(* CODESYS project Elevator.ecp

Project tree, tasks and I/O mapping:
  Controller : 750-8214 PFC200 G2 2ETH RS CAN, WAGO, order no. 0750-8214, version 5.13.2.32
    application Application
      libraries: ; WagoAppPlcModbus, 1.1.2.3 (WAGO)
      task PLC_Task (cyclic, interval t#50ms, priority 15) calls ModbusTester, Heis2Test, VariableAssociation
      task VISU_TASK (cyclic, interval 100 ms, priority 15) calls VisuElems.Visu_Prg
      global variables GVL
      program ModbusTester [ST]
      MODBUS/
        data type typHeis1_tcp
        data type typHeis2_tcp
      global variables MODBUS
      program VariableAssociation [ST]
      program Heis2Test [ST]
      visualisation Visualization
    Kbus : Kbus, WAGO, version 1.4.0.2
        unmapped channels: K-BUS diagnostics
      _8_DI_Generic : 075x-8DI, WAGO, order no. 075x-8DI, version 0.0.0.13
          settings: K-BUS Module slot index = 1
          unmapped channels: _IN
      _8_DO_Generic : 075x-8DO, WAGO, order no. 075x-8DO, version 0.0.0.13
          settings: K-BUS Module slot index = 2
          unmapped channels: _OUT
    MODBUS
      MODBUS : MODBUS, WAGO, order no. n/a, version 1.1.1.15
        _internal_1006_0001_Master : MODBUS Master, WAGO, order no. n/a, version 1.1.1.15
          _internal_1006_0001_IP : MODBUS IP Interface, WAGO, order no. n/a, version 1.1.1.15
              settings: IP settings.Address = '192.168.0.3'
            Heis1_tcp : MODBUS Remote Slave, WAGO, order no. n/a, version 1.1.1.15
                settings: Channel100005.Priority = 1; Channel100005.Cycle Time = 200 ms; Channel100005.Read Length = 24 Registers or Coils; ChannelOffset100010 = 0; ChannelOffset100030 = 1; ChannelOffset100050 = 2; ChannelOffset100070 = 3; ChannelOffset100090 = 4; ChannelOffset100110 = 5; ChannelOffset100130 = 6; ChannelOffset100150 = 7; ChannelOffset100170 = 8; ChannelOffset100190 = 9; ChannelOffset100210 = 10; ChannelOffset100230 = 11; ChannelOffset100250 = 12; ChannelOffset100270 = 13; ChannelOffset100290 = 14; ChannelOffset100310 = 15; ChannelOffset100330 = 16; ChannelOffset100350 = 17; ChannelOffset100370 = 18; ChannelOffset100390 = 19; ChannelOffset100410 = 20; ChannelOffset100430 = 21; ChannelOffset100450 = 22; ChannelOffset100470 = 23; Channel100485.Priority = 1; Channel100485.Cycle Time = 200 ms; Channel100485.Write Address = 512 Registers or Coils; Channel100485.Write Length = 16 Registers or Coils; ChannelOffset100490 = 0; ChannelOffset100510 = 1; ChannelOffset100530 = 2; ChannelOffset100550 = 3; ChannelOffset100570 = 4; ChannelOffset100590 = 5; ChannelOffset100610 = 6; ChannelOffset100630 = 7; ChannelOffset100650 = 8;
                  ChannelOffset100670 = 9; ChannelOffset100690 = 10; ChannelOffset100710 = 11; ChannelOffset100730 = 12; ChannelOffset100750 = 13; ChannelOffset100770 = 14; ChannelOffset100790 = 15; Slave address / Unit identifier = 2
                input  Application.MODBUS.Heis1_tcp.dIn_1 : BOOL  // ChannelMapping100020
                input  Application.MODBUS.Heis1_tcp.dIn_2 : BOOL  // ChannelMapping100040
                input  Application.MODBUS.Heis1_tcp.dIn_3 : BOOL  // ChannelMapping100060
                input  Application.MODBUS.Heis1_tcp.dIn_4 : BOOL  // ChannelMapping100080
                input  Application.MODBUS.Heis1_tcp.dIn_5 : BOOL  // ChannelMapping100100
                input  Application.MODBUS.Heis1_tcp.dIn_6 : BOOL  // ChannelMapping100120
                input  Application.MODBUS.Heis1_tcp.dIn_7 : BOOL  // ChannelMapping100140
                input  Application.MODBUS.Heis1_tcp.dIn_8 : BOOL  // ChannelMapping100160
                input  Application.MODBUS.Heis1_tcp.dIn_9 : BOOL  // ChannelMapping100180
                input  Application.MODBUS.Heis1_tcp.dIn_10 : BOOL  // ChannelMapping100200
                input  Application.MODBUS.Heis1_tcp.dIn_11 : BOOL  // ChannelMapping100220
                input  Application.MODBUS.Heis1_tcp.dIn_12 : BOOL  // ChannelMapping100240
                input  Application.MODBUS.Heis1_tcp.dIn_13 : BOOL  // ChannelMapping100260
                input  Application.MODBUS.Heis1_tcp.dIn_14 : BOOL  // ChannelMapping100280
                input  Application.MODBUS.Heis1_tcp.dIn_15 : BOOL  // ChannelMapping100300
                input  Application.MODBUS.Heis1_tcp.dIn_16 : BOOL  // ChannelMapping100320
                input  Application.MODBUS.Heis1_tcp.dIn_17 : BOOL  // ChannelMapping100340
                input  Application.MODBUS.Heis1_tcp.dIn_18 : BOOL  // ChannelMapping100360
                input  Application.MODBUS.Heis1_tcp.dIn_19 : BOOL  // ChannelMapping100380
                input  Application.MODBUS.Heis1_tcp.dIn_20 : BOOL  // ChannelMapping100400
                input  Application.MODBUS.Heis1_tcp.dIn_21 : BOOL  // ChannelMapping100420
                input  Application.MODBUS.Heis1_tcp.dIn_22 : BOOL  // ChannelMapping100440
                input  Application.MODBUS.Heis1_tcp.dIn_23 : BOOL  // ChannelMapping100460
                input  Application.MODBUS.Heis1_tcp.dIn_24 : BOOL  // ChannelMapping100480
                output Application.MODBUS.Heis1_tcp.dOut_1 : BOOL  // ChannelMapping100500
                output Application.MODBUS.Heis1_tcp.dOut_2 : BOOL  // ChannelMapping100520
                output Application.MODBUS.Heis1_tcp.dOut_3 : BOOL  // ChannelMapping100540
                output Application.MODBUS.Heis1_tcp.dOut_4 : BOOL  // ChannelMapping100560
                output Application.MODBUS.Heis1_tcp.dOut_5 : BOOL  // ChannelMapping100580
                output Application.MODBUS.Heis1_tcp.dOut_6 : BOOL  // ChannelMapping100600
                output Application.MODBUS.Heis1_tcp.dOut_7 : BOOL  // ChannelMapping100620
                output Application.MODBUS.Heis1_tcp.dOut_8 : BOOL  // ChannelMapping100640
                output Application.MODBUS.Heis1_tcp.dOut_9 : BOOL  // ChannelMapping100660
                output Application.MODBUS.Heis1_tcp.dOut_10 : BOOL  // ChannelMapping100680
                output Application.MODBUS.Heis1_tcp.dOut_11 : BOOL  // ChannelMapping100700
                output Application.MODBUS.Heis1_tcp.dOut_12 : BOOL  // ChannelMapping100720
                output Application.MODBUS.Heis1_tcp.dOut_13 : BOOL  // ChannelMapping100740
                output Application.MODBUS.Heis1_tcp.dOut_14 : BOOL  // ChannelMapping100760
                output Application.MODBUS.Heis1_tcp.dOut_15 : BOOL  // ChannelMapping100780
                output Application.MODBUS.Heis1_tcp.dOut_16 : BOOL  // ChannelMapping100800
          _internal_1006_0001_IP_1 : MODBUS IP Interface, WAGO, order no. n/a, version 1.1.1.15
              settings: IP settings.Address = '192.168.0.4'
            Heis2_tcp : MODBUS Remote Slave, WAGO, order no. n/a, version 1.1.1.15
                settings: Channel100005.Priority = 1; Channel100005.Cycle Time = 200 ms; Channel100005.Read Length = 24 Registers or Coils; ChannelOffset100010 = 0; ChannelOffset100030 = 1; ChannelOffset100050 = 2; ChannelOffset100070 = 3; ChannelOffset100090 = 4; ChannelOffset100110 = 5; ChannelOffset100130 = 6; ChannelOffset100150 = 7; ChannelOffset100170 = 8; ChannelOffset100190 = 9; ChannelOffset100210 = 10; ChannelOffset100230 = 11; ChannelOffset100250 = 12; ChannelOffset100270 = 13; ChannelOffset100290 = 14; ChannelOffset100310 = 15; ChannelOffset100330 = 16; ChannelOffset100350 = 17; ChannelOffset100370 = 18; ChannelOffset100390 = 19; ChannelOffset100410 = 20; ChannelOffset100430 = 21; ChannelOffset100450 = 22; ChannelOffset100470 = 23; Channel100485.Priority = 1; Channel100485.Cycle Time = 200 ms; Channel100485.Write Address = 512 Registers or Coils; Channel100485.Write Length = 16 Registers or Coils; ChannelOffset100490 = 0; ChannelOffset100510 = 1; ChannelOffset100530 = 2; ChannelOffset100550 = 3; ChannelOffset100570 = 4; ChannelOffset100590 = 5; ChannelOffset100610 = 6; ChannelOffset100630 = 7; ChannelOffset100650 = 8;
                  ChannelOffset100670 = 9; ChannelOffset100690 = 10; ChannelOffset100710 = 11; ChannelOffset100730 = 12; ChannelOffset100750 = 13; ChannelOffset100770 = 14; ChannelOffset100790 = 15; Slave address / Unit identifier = 2
                input  Application.MODBUS.Heis2_tcp.dIn_1 : BOOL  // ChannelMapping100020
                input  Application.MODBUS.Heis2_tcp.dIn_2 : BOOL  // ChannelMapping100040
                input  Application.MODBUS.Heis2_tcp.dIn_3 : BOOL  // ChannelMapping100060
                input  Application.MODBUS.Heis2_tcp.dIn_4 : BOOL  // ChannelMapping100080
                input  Application.MODBUS.Heis2_tcp.dIn_5 : BOOL  // ChannelMapping100100
                input  Application.MODBUS.Heis2_tcp.dIn_6 : BOOL  // ChannelMapping100120
                input  Application.MODBUS.Heis2_tcp.dIn_7 : BOOL  // ChannelMapping100140
                input  Application.MODBUS.Heis2_tcp.dIn_8 : BOOL  // ChannelMapping100160
                input  Application.MODBUS.Heis2_tcp.dIn_9 : BOOL  // ChannelMapping100180
                input  Application.MODBUS.Heis2_tcp.dIn_10 : BOOL  // ChannelMapping100200
                input  Application.MODBUS.Heis2_tcp.dIn_11 : BOOL  // ChannelMapping100220
                input  Application.MODBUS.Heis2_tcp.dIn_12 : BOOL  // ChannelMapping100240
                input  Application.MODBUS.Heis2_tcp.dIn_13 : BOOL  // ChannelMapping100260
                input  Application.MODBUS.Heis2_tcp.dIn_14 : BOOL  // ChannelMapping100280
                input  Application.MODBUS.Heis2_tcp.dIn_15 : BOOL  // ChannelMapping100300
                input  Application.MODBUS.Heis2_tcp.dIn_16 : BOOL  // ChannelMapping100320
                input  Application.MODBUS.Heis2_tcp.dIn_17 : BOOL  // ChannelMapping100340
                input  Application.MODBUS.Heis2_tcp.dIn_18 : BOOL  // ChannelMapping100360
                input  Application.MODBUS.Heis2_tcp.dIn_19 : BOOL  // ChannelMapping100380
                input  Application.MODBUS.Heis2_tcp.dIn_20 : BOOL  // ChannelMapping100400
                input  Application.MODBUS.Heis2_tcp.dIn_21 : BOOL  // ChannelMapping100420
                input  Application.MODBUS.Heis2_tcp.dIn_22 : BOOL  // ChannelMapping100440
                input  Application.MODBUS.Heis2_tcp.dIn_23 : BOOL  // ChannelMapping100460
                input  Application.MODBUS.Heis2_tcp.dIn_24 : BOOL  // ChannelMapping100480
                output Application.MODBUS.Heis2_tcp.dOut_1 : BOOL  // ChannelMapping100500
                output Application.MODBUS.Heis2_tcp.dOut_2 : BOOL  // ChannelMapping100520
                output Application.MODBUS.Heis2_tcp.dOut_3 : BOOL  // ChannelMapping100540
                output Application.MODBUS.Heis2_tcp.dOut_4 : BOOL  // ChannelMapping100560
                output Application.MODBUS.Heis2_tcp.dOut_5 : BOOL  // ChannelMapping100580
                output Application.MODBUS.Heis2_tcp.dOut_6 : BOOL  // ChannelMapping100600
                output Application.MODBUS.Heis2_tcp.dOut_7 : BOOL  // ChannelMapping100620
                output Application.MODBUS.Heis2_tcp.dOut_8 : BOOL  // ChannelMapping100640
                output Application.MODBUS.Heis2_tcp.dOut_9 : BOOL  // ChannelMapping100660
                output Application.MODBUS.Heis2_tcp.dOut_10 : BOOL  // ChannelMapping100680
                output Application.MODBUS.Heis2_tcp.dOut_11 : BOOL  // ChannelMapping100700
                output Application.MODBUS.Heis2_tcp.dOut_12 : BOOL  // ChannelMapping100720
                output Application.MODBUS.Heis2_tcp.dOut_13 : BOOL  // ChannelMapping100740
                output Application.MODBUS.Heis2_tcp.dOut_14 : BOOL  // ChannelMapping100760
                output Application.MODBUS.Heis2_tcp.dOut_15 : BOOL  // ChannelMapping100780
                output Application.MODBUS.Heis2_tcp.dOut_16 : BOOL  // ChannelMapping100800
    CANbus
    Common.PCI
    Serial
      COM1 : COM1, WAGO, version 0.0.0.19
  Heis1 : 750-352, WAGO, order no. 0750-0352, version 0.0.0.9
    Kbus : Kbus, WAGO, version 0.0.0.101
      _8_DI_Generic : 075x-8DI, WAGO, order no. 075x-8DI, version 0.0.0.13
          settings: K-BUS Module slot index = 1
          unmapped channels: _IN
      _8_DI_Generic_1 : 075x-8DI, WAGO, order no. 075x-8DI, version 0.0.0.13
          settings: K-BUS Module slot index = 2
          unmapped channels: _IN
      _8_DI_Generic_2 : 075x-8DI, WAGO, order no. 075x-8DI, version 0.0.0.13
          settings: K-BUS Module slot index = 3
          unmapped channels: _IN
      _8_DO_Generic : 075x-8DO, WAGO, order no. 075x-8DO, version 0.0.0.13
          settings: K-BUS Module slot index = 4
          unmapped channels: _OUT
      _8_DO_Generic_1 : 075x-8DO, WAGO, order no. 075x-8DO, version 0.0.0.13
          settings: K-BUS Module slot index = 5
          unmapped channels: _OUT
  Heis2 : 750-352, WAGO, order no. 0750-0352, version 0.0.0.9
    Kbus : Kbus, WAGO, version 0.0.0.101
      _8_DI_Generic : 075x-8DI, WAGO, order no. 075x-8DI, version 0.0.0.13
          settings: K-BUS Module slot index = 1
          unmapped channels: _IN
      _8_DI_Generic_1 : 075x-8DI, WAGO, order no. 075x-8DI, version 0.0.0.13
          settings: K-BUS Module slot index = 2
          unmapped channels: _IN
      _8_DI_Generic_2 : 075x-8DI, WAGO, order no. 075x-8DI, version 0.0.0.13
          settings: K-BUS Module slot index = 3
          unmapped channels: _IN
      _8_DO_Generic : 075x-8DO, WAGO, order no. 075x-8DO, version 0.0.0.13
          settings: K-BUS Module slot index = 4
          unmapped channels: _OUT
      _8_DO_Generic_1 : 075x-8DO, WAGO, order no. 075x-8DO, version 0.0.0.13
          settings: K-BUS Module slot index = 5
          unmapped channels: _OUT
  text list GlobalTextList
*)

// Controller/Application/MODBUS/typHeis1_tcp
TYPE typHeis1_tcp:
STRUCT
	dIn_1: BOOL;
	dIn_2: BOOL;
	dIn_3: BOOL;
	dIn_4: BOOL;
	dIn_5: BOOL;
	dIn_6: BOOL;
	dIn_7: BOOL;
	dIn_8: BOOL;
	dIn_9: BOOL;
	dIn_10: BOOL;
	dIn_11: BOOL;
	dIn_12: BOOL;
	dIn_13: BOOL;
	dIn_14: BOOL;
	dIn_15: BOOL;
	dIn_16: BOOL;
	dIn_17: BOOL;
	dIn_18: BOOL;
	dIn_19: BOOL;
	dIn_20: BOOL;
	dIn_21: BOOL;
	dIn_22: BOOL;
	dIn_23: BOOL;
	dIn_24: BOOL;
	dOut_1: BOOL;
	dOut_2: BOOL;
	dOut_3: BOOL;
	dOut_4: BOOL;
	dOut_5: BOOL;
	dOut_6: BOOL;
	dOut_7: BOOL;
	dOut_8: BOOL;
	dOut_9: BOOL;
	dOut_10: BOOL;
	dOut_11: BOOL;
	dOut_12: BOOL;
	dOut_13: BOOL;
	dOut_14: BOOL;
	dOut_15: BOOL;
	dOut_16: BOOL;
END_STRUCT
END_TYPE

// Controller/Application/MODBUS/typHeis2_tcp
TYPE typHeis2_tcp:
STRUCT
	dIn_1: BOOL;
	dIn_2: BOOL;
	dIn_3: BOOL;
	dIn_4: BOOL;
	dIn_5: BOOL;
	dIn_6: BOOL;
	dIn_7: BOOL;
	dIn_8: BOOL;
	dIn_9: BOOL;
	dIn_10: BOOL;
	dIn_11: BOOL;
	dIn_12: BOOL;
	dIn_13: BOOL;
	dIn_14: BOOL;
	dIn_15: BOOL;
	dIn_16: BOOL;
	dIn_17: BOOL;
	dIn_18: BOOL;
	dIn_19: BOOL;
	dIn_20: BOOL;
	dIn_21: BOOL;
	dIn_22: BOOL;
	dIn_23: BOOL;
	dIn_24: BOOL;
	dOut_1: BOOL;
	dOut_2: BOOL;
	dOut_3: BOOL;
	dOut_4: BOOL;
	dOut_5: BOOL;
	dOut_6: BOOL;
	dOut_7: BOOL;
	dOut_8: BOOL;
	dOut_9: BOOL;
	dOut_10: BOOL;
	dOut_11: BOOL;
	dOut_12: BOOL;
	dOut_13: BOOL;
	dOut_14: BOOL;
	dOut_15: BOOL;
	dOut_16: BOOL;
END_STRUCT
END_TYPE

// Controller/Application/GVL
VAR_GLOBAL	
    //Elevator 1
    ELEVATOR1STATE : INT; //IF the elevator is coming from up or down ore from idle
	E1FLOORSTATE : REAL; //Which floor the elevator is in.
	E1MotorUp : BOOL;
	E1MotorDown : BOOL;
	E1MotorFast : BOOL;
	E1MotorSlow : BOOL;
	DoorS1 : BOOL; //Floor 1, door switch 
	DoorS2 : BOOL; //Floor 2, door switch 
	DoorS3 : BOOL; //Floor 3, door switch 
	DoorS4 : BOOL; //Floor 4, door switch 
	
    //Buttons outside elevator
    S5 : BOOL; //Elevator 1, floor 4, down button
	S6 : BOOL; //Elevator 1, Floor 3, up button
	S7 : BOOL; //Elevator 1, floor 3, down button
	S8 : BOOL; //Elevator 1, floor 2, up button
	S9 : BOOL; //Elevator 1, floor 2, down button
	S10 : BOOL; //Elevator 1, floor 1, up button
	
	//Signals from buttons outside elivator	
	S10UPSignal: BOOL;//Elevator 1, floor 1, button up signal
	S9DownSignal: BOOL; //Elevator 1, floor 2, button down signal
	S8UPSignal: BOOL; //Elevator 1, floor 2, button up signal
	S7DownSignal: BOOL;//Elevator 1, floor 3, button down signal
	S6UpSignal: BOOL; //Elevator 1, floor 3, button up signal
	S5DownSignal: BOOL; //Elevator 1, floor 4, button down signal
	
	//Buttons inside elevator 1
	S11 : BOOL; //Elevator 1, button 1 in elevator
	S12 : BOOL; //Elevator 1, button 2 in elevator
	S13 : BOOL; //Elevator 1, button 2 in elevator
	S14 : BOOL; //Elevator 1, button 2 in elevator
	S15 : BOOL; //Alarm button
	
	//Buttons inside elivator
	S11Signal : BOOL;//Elevator 1, button 1 in elevator
	S12Signal : BOOL;//Elevator 1, button 2 in elevator	
	S13Signal : BOOL;//Elevator 1, button 3 in elevator
	S14Signal : BOOL;//Elevator 1, button 4 in elevator
    
	//Lamps
	//Inside
	E1H1 : BOOL; //Button 1 lamp
	E1H2 : BOOL; //Button 2 lamp
	E1H3 : BOOL; //Button 3 lamp
	E1H4 : BOOL; //Button 4 lamp	
	E1H16 : BOOL; //Alarm lamp
	//Outside
	E1H10 : BOOL; //Floor 4, down button lamp
	E1H11 : BOOL; //FLoor 3, up button lamp
	E1H12 : BOOL; //FLoor 3, down button lamp
	E1H13 : BOOL; //Floor 2, up button lamp
	E1H14 : BOOL; //FLoor 2, down button lamp
	E1H15 : BOOL; //FLoor 1, up button lamp
	
	//Sensors
	E1B1 : BOOL; //Fourth floor
	E1B2 : BOOL; //Fourth floor bottom
	E1B3 : BOOL; //Third floor top
	E1B4 : BOOL; //Third floor
	E1B5 : BOOL; //Third floor bottom
	E1B6 : BOOL; //Second floor top
	E1B7 : BOOL; //Second floor
	E1B8 : BOOL; //Second floor bottom
	E1B9 : BOOL; //First floor top
	E1B10 : BOOL; //First floor
	
	
	//Elevator 2
	ELEVATOR2STATE : INT; //IF the elevator is coming from up or down ore from idle
	E2FLOORSTATE : REAL; //Which floor the elevator is in.
	E2MotorUp : BOOL;  //Run motor upward
	E2MotorDown : BOOL; //Run motor downward
    
    //Buttons inside elevator 2
    S1 : BOOL; //Elevator 2, button 1 in elevator
	S2 : BOOL; //Elevator 2, button 2 in elevator
	S3 : BOOL; //Elevator 2, button 3 in elevator
	S4 : BOOL; //Elevator 2, button 4 in elevator
	
	//Buttons in elevator
    S1Signal : BOOL; //Elevator 2, button 1 signal in elevator
	S2Signal : BOOL; //Elevator 2, button 2 signal in elevator
	S3Signal : BOOL; //Elevator 2, button 3 signalin elevator
	S4Signal : BOOL; //Elevator 2, button  signalin elevator
	
	//Buttons outside Elevator 2
	S1Up : BOOL; //Elevator 2, Floor 1, button up
	S2Down : BOOL; //Elevator 2, floor 2 button down
	S2Up : BOOL; //Elevator 2, floor 2, button up
	S3Down : BOOL; //Elevator 2, floor 3, button down
	S3Up : BOOL; //Elevator 2, floor 3, button up
	S4Down : BOOL;	//Elevator 2, floor 4, button down
	SAlarm : BOOL; //Elevator 2, alarm button
	SEmergency : BOOL; //EmergencyStop

    //Buttons outside elevator
	S1UPSignal: BOOL;
	S2DownSignal: BOOL;
	S2UPSignal: BOOL;
	S3DownSignal: BOOL;
	S3UPSignal: BOOL;
	S4DownSignal: BOOL;
	
    //Lamps inside
	E2H1 : BOOL; //Elevator 2, button 1 light
	E2H2 : BOOL; //Elevator 2, button 2 light
	E2H3 : BOOL; //Elevator 2, Button 3 light
	E2H4 : BOOL; //Elevator 2, button 4 light 
	
	//Lamps outside
	E2H5 : BOOL; //Elevator 2, floor 4 Light
	E2H6 : BOOL; //Elevator 2, fLoor 3 light
	E2H7 : BOOL; //Elevator 2, fLoor 2 light
	E2H8 : BOOL; //Elevator 2, floor 1 light
	
	//Sensors
	E2B1 : BOOL; //Elevator 2, first floor final
	E2B2 : BOOL; //Elevator 2, first floor
	E2B3 : BOOL; //Elevator 2, second floor
	E2B4 : BOOL; //Elevator 2, third floor
	E2B5 : BOOL; //Elevator 2, fourth floor
	E2B6 : BOOL; //Elevator 2, fourth floor final
	
END_VAR

// Controller/Application/MODBUS
{attribute 'qualified_only'}
VAR_GLOBAL
	Heis1_tcp: typHeis1_tcp;
	Heis2_tcp: typHeis2_tcp;
END_VAR

// Controller/Application/ModbusTester
PROGRAM ModbusTester
VAR
	stop : BOOL;
END_VAR

// Testprogram for the modbus conneciton
// Pressing the floor 3 down button will cause the elevator to drive up until it reaches floor 3.
// Pressing the floor 2 up button will cause the elevator to drive down until it reaches floor 2.

IF GVL.E1B1 THEN
	GVL.E1MotorUp := FALSE;
END_IF

IF GVL.E1B10 THEN
	E1MotorDown := FALSE;
END_IF

IF GVL.E1B7 THEN
	GVL.E1H13 := TRUE;
	ELSE GVL.E1H13 := FALSE;
END_IF

IF GVL.E1B4 THEN
	GVL.E1H12 := TRUE;
	ELSE GVL.E1H12 := FALSE;
END_IF

IF GVL.S8 AND NOT GVL.E1MotorUp AND NOT GVL.E1B7 THEN
	stop := FALSE;
	GVL.E1MotorDown := TRUE;
END_IF

IF GVL.E1MotorDown AND GVL.E1B6 THEN
		stop := TRUE;
END_IF

IF GVL.E1H12 AND NOT GVL.E1MotorDown AND NOT GVL.E1B4 THEN
	stop := FALSE;	
	GVL.E1MotorUp := TRUE;
END_IF

IF GVL.E1MotorUp AND GVL.E1B5 THEN
		stop := TRUE;
END_IF

IF stop THEN
	GVL.E1MotorUp := FALSE;
	GVL.E1MotorDown := FALSE;
END_IF

END_PROGRAM

// Controller/Application/Heis2Test
PROGRAM Heis2Test
VAR
	stop : BOOL;
END_VAR

IF GVL.E2B6 THEN
	E2MotorUp := FALSE;
END_IF

IF GVL.E2B1 THEN
	GVL.E2MotorDown := FALSE;
END_IF

IF GVL.E2B3 THEN
	GVL.E2H7 := TRUE;
	ELSE GVL.E2H7 := FALSE;
END_IF

IF GVL.E2B4 THEN
	GVL.E2H6 := TRUE;
	ELSE GVL.E2H6 := FALSE;
END_IF

IF GVL.S2Up AND NOT GVL.E2MotorUp AND NOT GVL.E2B3 THEN
	stop := FALSE;
	GVL.E2MotorDown := TRUE;
END_IF

IF GVL.E2MotorDown AND GVL.E2B3 THEN
		stop := TRUE;
END_IF

IF GVL.S3Down AND NOT GVL.E2MotorDown AND NOT GVL.E2B4 THEN
	stop := FALSE;	
	GVL.E2MotorUp := TRUE;
END_IF

IF GVL.E2MotorUp AND GVL.E2B4 THEN
		stop := TRUE;
END_IF

IF stop THEN
	GVL.E2MotorUp := FALSE;
	GVL.E2MotorDown := FALSE;
END_IF

END_PROGRAM

// Controller/Application/VariableAssociation
PROGRAM VariableAssociation
VAR
	
END_VAR

//Elevator 1
//Motor
MODBUS.Heis1_tcp.dOut_14 := E1MotorUp;
MODBUS.Heis1_tcp.dOut_16 := E1MotorDown;
MODBUS.Heis1_tcp.dOut_6 := E1MotorFast;
MODBUS.Heis1_tcp.dOut_4 := E1MotorSlow;

//Sensors
//Floor
GVL.E1B10 := MODBUS.Heis1_tcp.dIn_11;	//First floor 
GVL.E1B9 := MODBUS.Heis1_tcp.dIn_9;		//First floor top
GVL.E1B8 := MODBUS.Heis1_tcp.dIn_8;		//Second floor bottom
GVL.E1B7 := MODBUS.Heis1_tcp.dIn_6; 	//Second floor
GVL.E1B6 := MODBUS.Heis1_tcp.dIn_4;     //Second floor top
GVL.E1B5 := MODBUS.Heis1_tcp.dIn_2;		//Third floor bottom
GVL.E1B4 := MODBUS.Heis1_tcp.dIn_7; 	//Third floor
GVL.E1B3 := MODBUS.Heis1_tcp.dIn_5;		//Third floor top
GVL.E1B2 := MODBUS.Heis1_tcp.dIn_3;		//Fourth floor bottom
GVL.E1B1 := MODBUS.Heis1_tcp.dIn_1;		//Fourth floor

//Door
GVL.DoorS1 := MODBUS.Heis1_tcp.dIn_22; //Universal door sensor

//Call buttons
GVL.S10 := MODBUS.Heis1_tcp.dIn_17; // Up first floor
GVL.S9 := MODBUS.Heis1_tcp.dIn_16; // Down second floor
GVL.S8 := MODBUS.Heis1_tcp.dIn_14; //Up second floor
GVL.S7 := MODBUS.Heis1_tcp.dIn_12; //Down third floor
GVL.S6 := MODBUS.Heis1_tcp.dIn_10; //Up third floor
GVL.S5 := MODBUS.Heis1_tcp.dIn_15; //Down fourth floor

// Call lights
MODBUS.Heis1_tcp.dOut_12 := GVL.E1H10; // Down fourth floor
MODBUS.Heis1_tcp.dOut_10 := GVL.E1H11; //Up third floor
MODBUS.Heis1_tcp.dOut_15 := GVL.E1H12; //Down third floor
MODBUS.Heis1_tcp.dOut_13 := GVL.E1H13; //Up second floor
MODBUS.Heis1_tcp.dOut_11 := GVL.E1H14; //Down second floor
MODBUS.Heis1_tcp.dOut_9 := GVL.E1H15; //Up first floor

//Control board
//Buttons
GVL.S14 := MODBUS.Heis1_tcp.dIn_18; //Fourth floor
GVL.S13 := MODBUS.Heis1_tcp.dIn_23; //Third floor
GVL.S12 := MODBUS.Heis1_tcp.dIn_21; //Second floor
GVL.S11 := MODBUS.Heis1_tcp.dIn_19; //First floor;
GVL.S15 := MODBUS.Heis1_tcp.dIn_20; //Alarm button

//Lights
MODBUS.Heis1_tcp.dOut_1 := GVl.E1H1; // First floor lamp
MODBUS.Heis1_tcp.dOut_3 := GVL.E1H2; // Second floor lamp
MODBUS.Heis1_tcp.dOut_5 := GVL.E1H3; // Third floor lamp
MODBUS.Heis1_tcp.dOut_7 := GVL.E1H4; // Fourth floor lamp
MODBUS.Heis1_tcp.dOut_2 := GVL.E1H16; //Alarm lamp


//Elevator 2
//Motor
MODBUS.Heis2_tcp.dOut_1 := E2MotorUp; //Run motor upward
MODBUS.Heis2_tcp.dOut_3 := E2MotorDown; //Run motor downward

//Sensors
GVL.E2B1 := MODBUS.Heis2_tcp.dIn_19; // First floor final stop
GVL.E2B2 := MODBUS.Heis2_tcp.dIn_15; // First floor stop
GVL.E2B3 := MODBUS.Heis2_tcp.dIn_10; // Second floor stop
GVL.E2B4 := MODBUS.Heis2_tcp.dIn_12; // Third floor stop
GVL.E2B5 := MODBUS.Heis2_tcp.dIn_14; // Fourth floor stop
GVL.E2B6 := MODBUS.Heis2_tcp.dIn_16; // Fourth floor final stop

//Call buttons
GVL.S1Up := MODBUS.Heis2_tcp.dIn_1; // Up first floor
GVL.S2Down := MODBUS.Heis2_tcp.dIn_3; // Down second floor
GVL.S2Up := MODBUS.Heis2_tcp.dIn_5; // Up second floor
GVL.S3Down := MODBUS.Heis2_tcp.dIn_7; // Down third floor
GVL.S3Up := MODBUS.Heis2_tcp.dIn_2; // Up third floor
GVL.S4Down := MODBUS.Heis2_tcp.dIn_4; // Down fourth floor

//Call lights
MODBUS.Heis2_tcp.dOut_5 := GVL.E2H1; // First floor
MODBUS.Heis2_tcp.dOut_7 := GVL.E2H2; // Second floor
MODBUS.Heis2_tcp.dOut_2 := GVL.E2H3; // Third floor
MODBUS.Heis2_tcp.dOut_4 := GVL.E2H4; // Fourth floor

//Control board
//Buttons
GVL.S1 := MODBUS.Heis2_tcp.dIn_6; // First floor
GVL.S2 := MODBUS.Heis2_tcp.dIn_8; // Second floor
GVL.S3 := MODBUS.Heis2_tcp.dIn_9; // Third floor
GVL.S4 := MODBUS.Heis2_tcp.dIn_11; // Fourth floor
GVL.SAlarm := MODBUS.Heis2_tcp.dIn_17; //Alarm button
GVL.SEmergency := MODBUS.Heis2_tcp.dIn_13; //Emergency stop

//Lights
MODBUS.Heis2_tcp.dOut_6 := GVL.E2H8; // First floor
MODBUS.Heis2_tcp.dOut_8 := GVL.E2H7; // Second floor
MODBUS.Heis2_tcp.dOut_9 := GVL.E2H6; // Third floor
MODBUS.Heis2_tcp.dOut_11 := GVL.E2H5; // Fourth floor

END_PROGRAM

// Controller/Application/Visualization
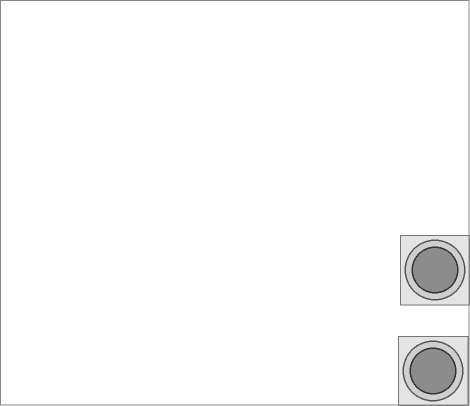
VISUALIZATION Visualization  // 470x406
    PushSwitch (400,235 70x70), variable: GVL.E2MotorUp, behaviour: TOGGLE, style: Switch-PushSwitch-Gray
    PushSwitch (398,336 70x70), variable: GVL.E2MotorDown, behaviour: TOGGLE, style: Switch-PushSwitch-Gray
END_VISUALIZATION
